(* IEC 61131-3 sources: Bob/Head_Pkg/ValveControl, 14 files *)

(* ---- Types.typ ---- *)
TYPE
	localValve_typ : 	STRUCT
		valveName : STRING[80];
		outputModuleOk : BOOL; (*variable to be linked to the module ok on the IO module used for the outputs*)
		inputModuleOk : BOOL; (*variable to be linked to the module ok on the IO module used for the inputs*)
		doOpen : BOOL; (*variable to be linked to the digital output which opens the valve*)
		doClose : BOOL; (*variable to be linked to the digital output which closes the valve*)
		diOpened : BOOL; (*variable to be linked to the digital input which indicates that the valve is opened*)
		diClosed : BOOL; (*variable to be linked to the digital input which indicates that the valve is closed*)
		position : INT;
		openDebounceTimer : TON;
		closeDebounceTimer : TON;
		openErrorTimer : TON;
		closeErrorTimer : TON;
		MpRecipeRegPar_0 : MpRecipeRegPar;
		MpRecipeRegPar_1 : MpRecipeRegPar;
		openError_r_trig : r_trig;
		closeError_r_trig : r_trig;
		open_and_close_error_r_trig : r_trig;
		io_error_r_trig : r_trig;
		io_error_f_trig : f_trig;
		openAndCloseAlarmID : UDINT;
		closeAlarmID : UDINT;
		openAlarmID : UDINT;
		alarmID : UDINT;
		moduleOKAlarmID : UDINT;
		powerOnTimer : TON;
	END_STRUCT;
END_TYPE

(* ---- balanceTankValve.st ---- *)
ACTION balanceTankAction:

    pCurrentValve ACCESS ADR(gModules[currentModule].heads[currentHead].balanceTank);
    pLocalValve ACCESS ADR(balanceTankValve[indexOf(currentModule, currentHead, NUM_OF_HEADS_PER_MODULE)]);

	IF (pCurrentValve.parameters.machineData.enabled = TRUE) THEN
		IF (pCurrentValve.status.errorActive <> TRUE) THEN

			IF (((pCurrentValve.commands.open = TRUE) AND (pCurrentValve.commands.close = FALSE)) AND
				(pLocalValve.doOpen = FALSE)) THEN
				logDebug(pLocalValve.valveName, 'Module %h, Head %h, Open Command', ADR(logArguments));
				pLocalValve.doOpen := TRUE;
				pLocalValve.doClose := FALSE;
			END_IF

			IF (((pCurrentValve.commands.close = TRUE) AND (pCurrentValve.commands.open = FALSE)) AND
				(pLocalValve.doClose = FALSE)) THEN
				logDebug(pLocalValve.valveName, 'Module %h, Head %h, Close Command', ADR(logArguments));
				pLocalValve.doClose := TRUE;
				pLocalValve.doOpen := FALSE;
			END_IF

			IF (((pCurrentValve.commands.close = FALSE) AND (pCurrentValve.commands.open = FALSE)) AND
				((pLocalValve.doClose <> FALSE) OR (pLocalValve.doOpen <> FALSE))) THEN
				logDebug(pLocalValve.valveName, 'Module %h, Head %h, Center Command', ADR(logArguments));
				pLocalValve.doClose := FALSE;
				pLocalValve.doOpen := FALSE;
			END_IF

		END_IF

		checkValveAlarms;
        updateValveState;

		// 20ms debounce timer
		pLocalValve.openDebounceTimer.IN    := pLocalValve.diOpened;
		pLocalValve.openDebounceTimer.PT    := pCurrentValve.parameters.machineData.debounceTime;
		pLocalValve.openDebounceTimer();

		// 20ms debounce timer
		pLocalValve.closeDebounceTimer.IN := pLocalValve.diClosed;
		pLocalValve.closeDebounceTimer.PT := pCurrentValve.parameters.machineData.debounceTime;
		pLocalValve.closeDebounceTimer();

		pCurrentValve.status.opened             := pLocalValve.openDebounceTimer.Q;
		pCurrentValve.status.closed             := pLocalValve.closeDebounceTimer.Q;
		pCurrentValve.status.centered           := ((pCurrentValve.status.opened <> TRUE) AND (pCurrentValve.status.closed <> TRUE));
		pCurrentValve.status.position           := 0;
		pCurrentValve.status.fullFlowAchieved   := FALSE;

        handleValveErrors;

    END_IF

END_ACTION

(* ---- counterStretchRodValve.st ---- *)
ACTION counterStretchRodAction:

    pCurrentValve ACCESS ADR(gModules[currentModule].heads[currentHead].counterStretchRod );
    pLocalValve ACCESS ADR(counterStretchRodValve[indexOf(currentModule, currentHead, NUM_OF_HEADS_PER_MODULE)]);

	IF (pCurrentValve.parameters.machineData.enabled = TRUE) THEN

		IF (pCurrentValve.status.errorActive <> TRUE) THEN

			IF (((pCurrentValve.commands.open = TRUE) AND (pCurrentValve.commands.close = FALSE)) AND
				(pLocalValve.doOpen = FALSE)) THEN
				logDebug(pLocalValve.valveName, 'Module %h, Head %h, Open Command', ADR(logArguments));
				pLocalValve.doOpen := TRUE;
				pLocalValve.doClose := FALSE;
			END_IF

			IF (((pCurrentValve.commands.close = TRUE) AND (pCurrentValve.commands.open = FALSE)) AND
				(pLocalValve.doClose = FALSE)) THEN
				logDebug(pLocalValve.valveName, 'Module %h, Head %h, Close Command', ADR(logArguments));
				pLocalValve.doClose := TRUE;
				pLocalValve.doOpen := FALSE;
			END_IF

			IF (((pCurrentValve.commands.close = FALSE) AND (pCurrentValve.commands.open = FALSE)) AND
				((pLocalValve.doClose <> FALSE) OR (pLocalValve.doOpen <> FALSE))) THEN
				logDebug(pLocalValve.valveName, 'Module %h, Head %h, Center Command', ADR(logArguments));
				pLocalValve.doClose := FALSE;
				pLocalValve.doOpen := FALSE;
			END_IF

		END_IF

		checkValveAlarms;
        updateValveState;

        // 20ms debounce timer
		pLocalValve.openDebounceTimer.IN    := pLocalValve.diOpened;
		pLocalValve.openDebounceTimer.PT    := pCurrentValve.parameters.machineData.debounceTime;
		pLocalValve.openDebounceTimer();

		// 20ms debounce timer
		pLocalValve.closeDebounceTimer.IN := pLocalValve.diClosed;
		pLocalValve.closeDebounceTimer.PT := pCurrentValve.parameters.machineData.debounceTime;
		pLocalValve.closeDebounceTimer();

		pCurrentValve.status.opened             := pLocalValve.openDebounceTimer.Q;
		pCurrentValve.status.closed             := pLocalValve.closeDebounceTimer.Q;
		pCurrentValve.status.centered           := ((pCurrentValve.status.opened <> TRUE) AND (pCurrentValve.status.closed <> TRUE));
		pCurrentValve.status.position           := 0;
		pCurrentValve.status.fullFlowAchieved   := FALSE;

        handleValveErrors;

	END_IF

END_ACTION

(* ---- cylinderVentValve.st ---- *)
ACTION cylinderVentAction:

    pCurrentValve ACCESS ADR(gModules[currentModule].heads[currentHead].cylinderVent);
    pLocalValve ACCESS ADR(cylinderVentValve[indexOf(currentModule, currentHead, NUM_OF_HEADS_PER_MODULE)]);

	IF (pCurrentValve.parameters.machineData.enabled = TRUE) THEN

		IF (pCurrentValve.status.errorActive <> TRUE) THEN

			IF (((pCurrentValve.commands.open = TRUE) AND (pCurrentValve.commands.close = FALSE)) AND
				(pLocalValve.doOpen = FALSE)) THEN
				logDebug('Cylinder Vent Valve', 'Module %h, Head %h, Open Command', ADR(logArguments));
				pLocalValve.doOpen := TRUE;
				pLocalValve.doClose := FALSE;
			END_IF

			IF (((pCurrentValve.commands.close = TRUE) AND (pCurrentValve.commands.open = FALSE)) AND
				(pLocalValve.doClose = FALSE)) THEN
				logDebug('Cylinder Vent Valve', 'Module %h, Head %h, Close Command', ADR(logArguments));
				pLocalValve.doClose := TRUE;
				pLocalValve.doOpen := FALSE;
			END_IF

			IF (((pCurrentValve.commands.close = FALSE) AND (pCurrentValve.commands.open = FALSE)) AND
				((pLocalValve.doClose <> FALSE) OR (pLocalValve.doOpen <> FALSE))) THEN
				logDebug('Cylinder Vent Valve', 'Module %h, Head %h, Center Command', ADR(logArguments));
				pLocalValve.doClose := FALSE;
				pLocalValve.doOpen := FALSE;
			END_IF

		END_IF

        checkValveAlarms;
        updateValveState;

		// 20ms debounce timer
		pLocalValve.openDebounceTimer.IN    := pLocalValve.diOpened;
		pLocalValve.openDebounceTimer.PT    := pCurrentValve.parameters.machineData.debounceTime;
		pLocalValve.openDebounceTimer();

		// 20ms debounce timer
		pLocalValve.closeDebounceTimer.IN := pLocalValve.diClosed;
		pLocalValve.closeDebounceTimer.PT := pCurrentValve.parameters.machineData.debounceTime;
		pLocalValve.closeDebounceTimer();

		pCurrentValve.status.opened             := pLocalValve.openDebounceTimer.Q;
		pCurrentValve.status.closed             := pLocalValve.closeDebounceTimer.Q;
		pCurrentValve.status.centered           := ((pCurrentValve.status.opened <> TRUE) AND (pCurrentValve.status.closed <> TRUE));
		pCurrentValve.status.position           := 0;
		pCurrentValve.status.fullFlowAchieved   := FALSE;

        handleValveErrors;

	END_IF

END_ACTION

(* ---- fillLevelCylinderValve.st ---- *)
ACTION fillLevelCylinderValveAction:

    pCurrentValve ACCESS ADR(gModules[currentModule].heads[currentHead].fillLevelCylinderValve);
    pLocalValve ACCESS ADR(fillLevelCylinderValve[indexOf(currentModule, currentHead, NUM_OF_HEADS_PER_MODULE)]);

	IF (pCurrentValve.parameters.machineData.enabled = TRUE) THEN

		IF (pCurrentValve.status.errorActive <> TRUE) THEN

			IF (((pCurrentValve.commands.open = TRUE) AND (pCurrentValve.commands.close = FALSE)) AND
				(pLocalValve.doOpen = FALSE)) THEN
				logDebug(pLocalValve.valveName, 'Module %h, Head %h, Retract Command', ADR(logArguments));
				pLocalValve.doOpen := TRUE;
				pLocalValve.doClose := FALSE;
			END_IF

			IF (((pCurrentValve.commands.close = TRUE) AND (pCurrentValve.commands.open = FALSE)) AND
				(pLocalValve.doClose = FALSE)) THEN
				logDebug(pLocalValve.valveName, 'Module %h, Head %h, Extend Command', ADR(logArguments));
				pLocalValve.doClose := TRUE;
				pLocalValve.doOpen := FALSE;
			END_IF

			IF (((pCurrentValve.commands.close = FALSE) AND (pCurrentValve.commands.open = FALSE)) AND
				((pLocalValve.doClose <> FALSE) OR (pLocalValve.doOpen <> FALSE))) THEN
				logDebug(pLocalValve.valveName, 'Module %h, Head %h, Center Command', ADR(logArguments));
				pLocalValve.doClose := FALSE;
				pLocalValve.doOpen := FALSE;
			END_IF

		END_IF

        checkValveAlarms;
        updateValveState;

		// 20ms debounce timer
		pLocalValve.openDebounceTimer.IN    := pLocalValve.diOpened;
		pLocalValve.openDebounceTimer.PT    := pCurrentValve.parameters.machineData.debounceTime;
		pLocalValve.openDebounceTimer();

		// 20ms debounce timer
		pLocalValve.closeDebounceTimer.IN := pLocalValve.diClosed;
		pLocalValve.closeDebounceTimer.PT := pCurrentValve.parameters.machineData.debounceTime;
		pLocalValve.closeDebounceTimer();

		pCurrentValve.status.opened             := pLocalValve.openDebounceTimer.Q;
		pCurrentValve.status.closed             := pLocalValve.closeDebounceTimer.Q;
		pCurrentValve.status.centered           := ((pCurrentValve.status.opened <> TRUE) AND (pCurrentValve.status.closed <> TRUE));
		pCurrentValve.status.position           := 0;
		pCurrentValve.status.fullFlowAchieved   := FALSE;

        handleValveErrors;

	END_IF

END_ACTION

(* ---- fillLevelDrainValve.st ---- *)
ACTION fillLevelDrainValveAction:

    pCurrentValve ACCESS ADR(gModules[currentModule].heads[currentHead].fillLevelDrainValve);
    pLocalValve ACCESS ADR(fillLevelDrainValve[indexOf(currentModule, currentHead, NUM_OF_HEADS_PER_MODULE)]);

	IF (pCurrentValve.parameters.machineData.enabled = TRUE) THEN

		IF (pCurrentValve.status.errorActive <> TRUE) THEN

			IF (((pCurrentValve.commands.open = TRUE) AND (pCurrentValve.commands.close = FALSE)) AND
				(pLocalValve.doOpen = FALSE)) THEN
				logDebug(pLocalValve.valveName, 'Module %h, Head %h, Open Command', ADR(logArguments));
				pLocalValve.doOpen := TRUE;
				pLocalValve.doClose := FALSE;
			END_IF

			IF (((pCurrentValve.commands.close = TRUE) AND (pCurrentValve.commands.open = FALSE)) AND
				(pLocalValve.doClose = FALSE)) THEN
				logDebug(pLocalValve.valveName, 'Module %h, Head %h, Close Command', ADR(logArguments));
				pLocalValve.doClose := TRUE;
				pLocalValve.doOpen := FALSE;
			END_IF

			IF (((pCurrentValve.commands.close = FALSE) AND (pCurrentValve.commands.open = FALSE)) AND
				((pLocalValve.doClose <> FALSE) OR (pLocalValve.doOpen <> FALSE))) THEN
				logDebug(pLocalValve.valveName, 'Module %h, Head %h, Center Command', ADR(logArguments));
				pLocalValve.doClose := FALSE;
				pLocalValve.doOpen := FALSE;
			END_IF

		END_IF

        checkValveAlarms;
        updateValveState;

		// 20ms debounce timer
		pLocalValve.openDebounceTimer.IN    := pLocalValve.diOpened;
		pLocalValve.openDebounceTimer.PT    := pCurrentValve.parameters.machineData.debounceTime;
		pLocalValve.openDebounceTimer();

		// 20ms debounce timer
		pLocalValve.closeDebounceTimer.IN := pLocalValve.diClosed;
		pLocalValve.closeDebounceTimer.PT := pCurrentValve.parameters.machineData.debounceTime;
		pLocalValve.closeDebounceTimer();

		pCurrentValve.status.opened             := pLocalValve.openDebounceTimer.Q;
		pCurrentValve.status.closed             := pLocalValve.closeDebounceTimer.Q;
		pCurrentValve.status.centered           := ((pCurrentValve.status.opened <> TRUE) AND (pCurrentValve.status.closed <> TRUE));
		pCurrentValve.status.position           := 0;
		pCurrentValve.status.fullFlowAchieved   := FALSE;

        handleValveErrors;

	END_IF

END_ACTION

(* ---- fillLevelSuctionValve.st ---- *)
ACTION fillLevelSuctionValveAction:

    pCurrentValve ACCESS ADR(gModules[currentModule].heads[currentHead].fillLevelSuctionValve);
    pLocalValve ACCESS ADR(fillLevelSuctionValve[indexOf(currentModule, currentHead, NUM_OF_HEADS_PER_MODULE)]);

	IF (pCurrentValve.parameters.machineData.enabled = TRUE) THEN

		IF (pCurrentValve.status.errorActive <> TRUE) THEN

			IF (((pCurrentValve.commands.open = TRUE) AND (pCurrentValve.commands.close = FALSE)) AND
				(pLocalValve.doOpen = FALSE)) THEN
				logDebug(pLocalValve.valveName, 'Module %h, Head %h, Open Command', ADR(logArguments));
				pLocalValve.doOpen := TRUE;
				pLocalValve.doClose := FALSE;
			END_IF

			IF (((pCurrentValve.commands.close = TRUE) AND (pCurrentValve.commands.open = FALSE)) AND
				(pLocalValve.doClose = FALSE)) THEN
				logDebug(pLocalValve.valveName, 'Module %h, Head %h, Close Command', ADR(logArguments));
				pLocalValve.doClose := TRUE;
				pLocalValve.doOpen := FALSE;
			END_IF

			IF (((pCurrentValve.commands.close = FALSE) AND (pCurrentValve.commands.open = FALSE)) AND
				((pLocalValve.doClose <> FALSE) OR (pLocalValve.doOpen <> FALSE))) THEN
				logDebug(pLocalValve.valveName, 'Module %h, Head %h, Center Command', ADR(logArguments));
				pLocalValve.doClose := FALSE;
				pLocalValve.doOpen := FALSE;
			END_IF

        END_IF

        checkValveAlarms;
        updateValveState;

		// 20ms debounce timer
		pLocalValve.openDebounceTimer.IN    := pLocalValve.diOpened;
		pLocalValve.openDebounceTimer.PT    := pCurrentValve.parameters.machineData.debounceTime;
		pLocalValve.openDebounceTimer();

		// 20ms debounce timer
		pLocalValve.closeDebounceTimer.IN := pLocalValve.diClosed;
		pLocalValve.closeDebounceTimer.PT := pCurrentValve.parameters.machineData.debounceTime;
		pLocalValve.closeDebounceTimer();

		pCurrentValve.status.opened             := pLocalValve.openDebounceTimer.Q;
		pCurrentValve.status.closed             := pLocalValve.closeDebounceTimer.Q;
		pCurrentValve.status.centered           := ((pCurrentValve.status.opened <> TRUE) AND (pCurrentValve.status.closed <> TRUE));
		pCurrentValve.status.position           := 0;
		pCurrentValve.status.fullFlowAchieved   := FALSE;

        handleValveErrors;

	END_IF

END_ACTION

(* ---- fillValve.st ---- *)
ACTION fillAction:

	pCurrentValve ACCESS ADR(gModules[currentModule].heads[currentHead].fillValve);
	pLocalValve ACCESS ADR(fillValve[indexOf(currentModule, currentHead, NUM_OF_HEADS_PER_MODULE)]);

	IF (pCurrentValve.parameters.machineData.enabled = TRUE) THEN

		IF (pCurrentValve.status.errorActive <> TRUE) THEN

			IF (((pCurrentValve.commands.open = TRUE) AND (pCurrentValve.commands.close = FALSE)) AND
				(pLocalValve.doOpen = FALSE)) THEN
				logDebug(pLocalValve.valveName, 'Module %h, Head %h, Open Command', ADR(logArguments));
				pLocalValve.doOpen := TRUE;
				pLocalValve.doClose := FALSE;

			END_IF

			IF (((pCurrentValve.commands.close = TRUE) AND (pCurrentValve.commands.open = FALSE)) AND
				(pLocalValve.doClose = FALSE)) THEN
				logDebug(pLocalValve.valveName, 'Module %h, Head %h, Close Command', ADR(logArguments));
				pLocalValve.doClose := TRUE;
				pLocalValve.doOpen := FALSE;
			END_IF

			IF (((pCurrentValve.commands.close = FALSE) AND (pCurrentValve.commands.open = FALSE)) AND
				((pLocalValve.doClose <> FALSE) OR (pLocalValve.doOpen <> FALSE))) THEN
				logDebug(pLocalValve.valveName, 'Module %h, Head %h, Center Command', ADR(logArguments));
				pLocalValve.doClose := FALSE;
				pLocalValve.doOpen := FALSE;
			END_IF

		END_IF

        checkValveAlarms;
        updateValveState;

		// 20ms debounce timer
		pLocalValve.openDebounceTimer.IN    := pLocalValve.diOpened;
		pLocalValve.openDebounceTimer.PT    := pCurrentValve.parameters.machineData.debounceTime;
		pLocalValve.openDebounceTimer();

		// 20ms debounce timer
		pLocalValve.closeDebounceTimer.IN := pLocalValve.diClosed;
		pLocalValve.closeDebounceTimer.PT := pCurrentValve.parameters.machineData.debounceTime;
		pLocalValve.closeDebounceTimer();

		pCurrentValve.status.opened             := pLocalValve.openDebounceTimer.Q;
		pCurrentValve.status.closed             := pLocalValve.closeDebounceTimer.Q;
		pCurrentValve.status.centered           := ((pCurrentValve.status.opened <> TRUE) AND (pCurrentValve.status.closed <> TRUE));
		pCurrentValve.status.position           := 0;
		pCurrentValve.status.fullFlowAchieved   := FALSE;

        handleValveErrors;

	END_IF

END_ACTION

(* ---- formingValve.st ---- *)
ACTION formingValveAction:

    pCurrentValve ACCESS ADR(gModules[currentModule].heads[currentHead].formingValve);
    pLocalValve ACCESS ADR(formingValve[indexOf(currentModule, currentHead, NUM_OF_HEADS_PER_MODULE)]);

	IF (pCurrentValve.parameters.machineData.enabled = TRUE) THEN

		IF (pCurrentValve.status.errorActive <> TRUE) THEN

			IF (((pCurrentValve.commands.open = TRUE) AND (pCurrentValve.commands.close = FALSE)) AND
				(pLocalValve.doOpen = FALSE)) THEN
				logDebug(pLocalValve.valveName, 'Module %h, Head %h, Open Command', ADR(logArguments));
				pLocalValve.doOpen := TRUE;
				pLocalValve.doClose := FALSE;
			END_IF

			IF (((pCurrentValve.commands.close = TRUE) AND (pCurrentValve.commands.open = FALSE)) AND
				(pLocalValve.doClose = FALSE)) THEN
				logDebug(pLocalValve.valveName, 'Module %h, Head %h, Close Command', ADR(logArguments));
				pLocalValve.doClose := TRUE;
				pLocalValve.doOpen := FALSE;
			END_IF

			IF (((pCurrentValve.commands.close = FALSE) AND (pCurrentValve.commands.open = FALSE)) AND
				((pLocalValve.doClose <> FALSE) OR (pLocalValve.doOpen <> FALSE))) THEN
				logDebug(pLocalValve.valveName, 'Module %h, Head %h, Center Command', ADR(logArguments));
				pLocalValve.doClose := FALSE;
				pLocalValve.doOpen := FALSE;
			END_IF

		END_IF

        checkValveAlarms;
        updateValveState;

		// 20ms debounce timer
		pLocalValve.openDebounceTimer.IN    := pLocalValve.diOpened;
		pLocalValve.openDebounceTimer.PT    := pCurrentValve.parameters.machineData.debounceTime;
		pLocalValve.openDebounceTimer();

		// 20ms debounce timer
		pLocalValve.closeDebounceTimer.IN := pLocalValve.diClosed;
		pLocalValve.closeDebounceTimer.PT := pCurrentValve.parameters.machineData.debounceTime;
		pLocalValve.closeDebounceTimer();

		pCurrentValve.status.opened         := pLocalValve.openDebounceTimer.Q;
		pCurrentValve.status.closed         := pLocalValve.closeDebounceTimer.Q;
		pCurrentValve.status.centered       := ((pCurrentValve.status.opened <> TRUE) AND (pCurrentValve.status.closed <> TRUE));
		pCurrentValve.status.position       := 0;

        handleValveErrors;

	END_IF

END_ACTION

(* ---- Main.st ---- *)
PROGRAM _INIT

    // register the balance tank parameters
    gModules[0].heads[0].balanceTank;
    balanceTankValve[0].MpRecipeRegPar_0.PVName := ADR('gModules[0].heads[0].balanceTank.parameters.machineData');
    balanceTankValve[1].MpRecipeRegPar_0.PVName := ADR('gModules[0].heads[1].balanceTank.parameters.machineData');
    balanceTankValve[2].MpRecipeRegPar_0.PVName := ADR('gModules[1].heads[0].balanceTank.parameters.machineData');
    balanceTankValve[3].MpRecipeRegPar_0.PVName := ADR('gModules[1].heads[1].balanceTank.parameters.machineData');

    FOR currentHead:=0 TO NUMBER_OF_HEADS_M1 DO
        balanceTankValve[currentHead].MpRecipeRegPar_0.MpLink := ADR(gMachineRecipe);
        balanceTankValve[currentHead].MpRecipeRegPar_0.Enable := TRUE;
        balanceTankValve[currentHead].MpRecipeRegPar_0.Category := ADR(MACHINE_CATEGORY);
        balanceTankValve[currentHead].MpRecipeRegPar_0();
    END_FOR

    balanceTankValve[0].MpRecipeRegPar_1.PVName := ADR('gModules[0].heads[0].balanceTank.parameters.processData');
    balanceTankValve[1].MpRecipeRegPar_1.PVName := ADR('gModules[0].heads[1].balanceTank.parameters.processData');
    balanceTankValve[2].MpRecipeRegPar_1.PVName := ADR('gModules[1].heads[0].balanceTank.parameters.processData');
    balanceTankValve[3].MpRecipeRegPar_1.PVName := ADR('gModules[1].heads[1].balanceTank.parameters.processData');

    FOR currentHead:=0 TO NUMBER_OF_HEADS_M1 DO
        balanceTankValve[currentHead].MpRecipeRegPar_1.MpLink := ADR(gProcessRecipe);
        balanceTankValve[currentHead].MpRecipeRegPar_1.Enable := TRUE;
        balanceTankValve[currentHead].MpRecipeRegPar_1.Category := ADR(PROCESS_CATEGORY);
        balanceTankValve[currentHead].MpRecipeRegPar_1();
    END_FOR

    // register the fill valve parameters
    gModules[0].heads[0].fillValve;
    fillValve[0].MpRecipeRegPar_0.PVName := ADR('gModules[0].heads[0].fillValve.parameters.machineData');
    fillValve[1].MpRecipeRegPar_0.PVName := ADR('gModules[0].heads[1].fillValve.parameters.machineData');
    fillValve[2].MpRecipeRegPar_0.PVName := ADR('gModules[1].heads[0].fillValve.parameters.machineData');
    fillValve[3].MpRecipeRegPar_0.PVName := ADR('gModules[1].heads[1].fillValve.parameters.machineData');

    FOR currentHead:=0 TO NUMBER_OF_HEADS_M1 DO
        fillValve[currentHead].MpRecipeRegPar_0.MpLink := ADR(gMachineRecipe);
        fillValve[currentHead].MpRecipeRegPar_0.Enable := TRUE;
        fillValve[currentHead].MpRecipeRegPar_0.Category := ADR(MACHINE_CATEGORY);
        fillValve[currentHead].MpRecipeRegPar_0();
    END_FOR

    fillValve[0].MpRecipeRegPar_1.PVName := ADR('gModules[0].heads[0].fillValve.parameters.processData');
    fillValve[1].MpRecipeRegPar_1.PVName := ADR('gModules[0].heads[1].fillValve.parameters.processData');
    fillValve[2].MpRecipeRegPar_1.PVName := ADR('gModules[1].heads[0].fillValve.parameters.processData');
    fillValve[3].MpRecipeRegPar_1.PVName := ADR('gModules[1].heads[1].fillValve.parameters.processData');

    FOR currentHead:=0 TO NUMBER_OF_HEADS_M1 DO
        fillValve[currentHead].MpRecipeRegPar_1.MpLink := ADR(gProcessRecipe);
        fillValve[currentHead].MpRecipeRegPar_1.Enable := TRUE;
        fillValve[currentHead].MpRecipeRegPar_1.Category := ADR(PROCESS_CATEGORY);
        fillValve[currentHead].MpRecipeRegPar_1();
    END_FOR

    // register the fill vent parameters
    gModules[0].heads[0].cylinderVent;
    cylinderVentValve[0].MpRecipeRegPar_0.PVName := ADR('gModules[0].heads[0].cylinderVent.parameters.machineData');
    cylinderVentValve[1].MpRecipeRegPar_0.PVName := ADR('gModules[0].heads[1].cylinderVent.parameters.machineData');
    cylinderVentValve[2].MpRecipeRegPar_0.PVName := ADR('gModules[1].heads[0].cylinderVent.parameters.machineData');
    cylinderVentValve[3].MpRecipeRegPar_0.PVName := ADR('gModules[1].heads[1].cylinderVent.parameters.machineData');

    FOR currentHead:=0 TO NUMBER_OF_HEADS_M1 DO
        cylinderVentValve[currentHead].MpRecipeRegPar_0.MpLink := ADR(gMachineRecipe);
        cylinderVentValve[currentHead].MpRecipeRegPar_0.Enable := TRUE;
        cylinderVentValve[currentHead].MpRecipeRegPar_0.Category := ADR(MACHINE_CATEGORY);
        cylinderVentValve[currentHead].MpRecipeRegPar_0();
    END_FOR

    cylinderVentValve[0].MpRecipeRegPar_1.PVName := ADR('gModules[0].heads[0].cylinderVent.parameters.processData');
    cylinderVentValve[1].MpRecipeRegPar_1.PVName := ADR('gModules[0].heads[1].cylinderVent.parameters.processData');
    cylinderVentValve[2].MpRecipeRegPar_1.PVName := ADR('gModules[1].heads[0].cylinderVent.parameters.processData');
    cylinderVentValve[3].MpRecipeRegPar_1.PVName := ADR('gModules[1].heads[1].cylinderVent.parameters.processData');

    FOR currentHead:=0 TO NUMBER_OF_HEADS_M1 DO
        cylinderVentValve[currentHead].MpRecipeRegPar_1.MpLink := ADR(gProcessRecipe);
        cylinderVentValve[currentHead].MpRecipeRegPar_1.Enable := TRUE;
        cylinderVentValve[currentHead].MpRecipeRegPar_1.Category := ADR(PROCESS_CATEGORY);
        cylinderVentValve[currentHead].MpRecipeRegPar_1();
    END_FOR

    // register the nozzle parameters
    gModules[0].heads[0].nozzle;
    nozzleValve[0].MpRecipeRegPar_0.PVName := ADR('gModules[0].heads[0].nozzle.parameters.machineData');
    nozzleValve[1].MpRecipeRegPar_0.PVName := ADR('gModules[0].heads[1].nozzle.parameters.machineData');
    nozzleValve[2].MpRecipeRegPar_0.PVName := ADR('gModules[1].heads[0].nozzle.parameters.machineData');
    nozzleValve[3].MpRecipeRegPar_0.PVName := ADR('gModules[1].heads[1].nozzle.parameters.machineData');

    FOR currentHead:=0 TO NUMBER_OF_HEADS_M1 DO
        nozzleValve[currentHead].MpRecipeRegPar_0.MpLink := ADR(gMachineRecipe);
        nozzleValve[currentHead].MpRecipeRegPar_0.Enable := TRUE;
        nozzleValve[currentHead].MpRecipeRegPar_0.Category := ADR(MACHINE_CATEGORY);
        nozzleValve[currentHead].MpRecipeRegPar_0();
    END_FOR

    nozzleValve[0].MpRecipeRegPar_1.PVName := ADR('gModules[0].heads[0].nozzle.parameters.processData');
    nozzleValve[1].MpRecipeRegPar_1.PVName := ADR('gModules[0].heads[1].nozzle.parameters.processData');
    nozzleValve[2].MpRecipeRegPar_1.PVName := ADR('gModules[1].heads[0].nozzle.parameters.processData');
    nozzleValve[3].MpRecipeRegPar_1.PVName := ADR('gModules[1].heads[1].nozzle.parameters.processData');

    FOR currentHead:=0 TO NUMBER_OF_HEADS_M1 DO
        nozzleValve[currentHead].MpRecipeRegPar_1.MpLink := ADR(gProcessRecipe);
        nozzleValve[currentHead].MpRecipeRegPar_1.Enable := TRUE;
        nozzleValve[currentHead].MpRecipeRegPar_1.Category := ADR(PROCESS_CATEGORY);
        nozzleValve[currentHead].MpRecipeRegPar_1();
    END_FOR

    // register the recirculationValve parameters
    gModules[0].heads[0].recirculationValve;
    recirculationValve[0].MpRecipeRegPar_0.PVName := ADR('gModules[0].heads[0].recirculationValve.parameters.machineData');
    recirculationValve[1].MpRecipeRegPar_0.PVName := ADR('gModules[0].heads[1].recirculationValve.parameters.machineData');
    recirculationValve[2].MpRecipeRegPar_0.PVName := ADR('gModules[1].heads[0].recirculationValve.parameters.machineData');
    recirculationValve[3].MpRecipeRegPar_0.PVName := ADR('gModules[1].heads[1].recirculationValve.parameters.machineData');

    FOR currentHead:=0 TO NUMBER_OF_HEADS_M1 DO
        recirculationValve[currentHead].MpRecipeRegPar_0.MpLink := ADR(gMachineRecipe);
        recirculationValve[currentHead].MpRecipeRegPar_0.Enable := TRUE;
        recirculationValve[currentHead].MpRecipeRegPar_0.Category := ADR(MACHINE_CATEGORY);
        recirculationValve[currentHead].MpRecipeRegPar_0();
    END_FOR

    recirculationValve[0].MpRecipeRegPar_1.PVName := ADR('gModules[0].heads[0].recirculationValve.parameters.processData');
    recirculationValve[1].MpRecipeRegPar_1.PVName := ADR('gModules[0].heads[1].recirculationValve.parameters.processData');
    recirculationValve[2].MpRecipeRegPar_1.PVName := ADR('gModules[1].heads[0].recirculationValve.parameters.processData');
    recirculationValve[3].MpRecipeRegPar_1.PVName := ADR('gModules[1].heads[1].recirculationValve.parameters.processData');

    FOR currentHead:=0 TO NUMBER_OF_HEADS_M1 DO
        recirculationValve[currentHead].MpRecipeRegPar_1.MpLink := ADR(gProcessRecipe);
        recirculationValve[currentHead].MpRecipeRegPar_1.Enable := TRUE;
        recirculationValve[currentHead].MpRecipeRegPar_1.Category := ADR(PROCESS_CATEGORY);
        recirculationValve[currentHead].MpRecipeRegPar_1();
    END_FOR

    // register the sealPin parameters
    gModules[0].heads[0].sealPin;
    sealPinValve[0].MpRecipeRegPar_0.PVName := ADR('gModules[0].heads[0].sealPin.parameters.machineData');
    sealPinValve[1].MpRecipeRegPar_0.PVName := ADR('gModules[0].heads[1].sealPin.parameters.machineData');
    sealPinValve[2].MpRecipeRegPar_0.PVName := ADR('gModules[1].heads[0].sealPin.parameters.machineData');
    sealPinValve[3].MpRecipeRegPar_0.PVName := ADR('gModules[1].heads[1].sealPin.parameters.machineData');

    FOR currentHead:=0 TO NUMBER_OF_HEADS_M1 DO
        sealPinValve[currentHead].MpRecipeRegPar_0.MpLink := ADR(gMachineRecipe);
        sealPinValve[currentHead].MpRecipeRegPar_0.Enable := TRUE;
        sealPinValve[currentHead].MpRecipeRegPar_0.Category := ADR(MACHINE_CATEGORY);
        sealPinValve[currentHead].MpRecipeRegPar_0();
    END_FOR

    sealPinValve[0].MpRecipeRegPar_1.PVName := ADR('gModules[0].heads[0].sealPin.parameters.processData');
    sealPinValve[1].MpRecipeRegPar_1.PVName := ADR('gModules[0].heads[1].sealPin.parameters.processData');
    sealPinValve[2].MpRecipeRegPar_1.PVName := ADR('gModules[1].heads[0].sealPin.parameters.processData');
    sealPinValve[3].MpRecipeRegPar_1.PVName := ADR('gModules[1].heads[1].sealPin.parameters.processData');

    FOR currentHead:=0 TO NUMBER_OF_HEADS_M1 DO
        sealPinValve[currentHead].MpRecipeRegPar_1.MpLink := ADR(gProcessRecipe);
        sealPinValve[currentHead].MpRecipeRegPar_1.Enable := TRUE;
        sealPinValve[currentHead].MpRecipeRegPar_1.Category := ADR(PROCESS_CATEGORY);
        sealPinValve[currentHead].MpRecipeRegPar_1();
    END_FOR

    // register the sealPin parameters
    gModules[0].heads[0].sealPin;
    counterStretchRodValve[0].MpRecipeRegPar_0.PVName := ADR('gModules[0].heads[0].counterStretchRod.parameters.machineData');
    counterStretchRodValve[1].MpRecipeRegPar_0.PVName := ADR('gModules[0].heads[1].counterStretchRod.parameters.machineData');
    counterStretchRodValve[2].MpRecipeRegPar_0.PVName := ADR('gModules[1].heads[0].counterStretchRod.parameters.machineData');
    counterStretchRodValve[3].MpRecipeRegPar_0.PVName := ADR('gModules[1].heads[1].counterStretchRod.parameters.machineData');

    FOR currentHead:=0 TO NUMBER_OF_HEADS_M1 DO
        counterStretchRodValve[currentHead].MpRecipeRegPar_0.MpLink := ADR(gMachineRecipe);
        counterStretchRodValve[currentHead].MpRecipeRegPar_0.Enable := TRUE;
        counterStretchRodValve[currentHead].MpRecipeRegPar_0.Category := ADR(MACHINE_CATEGORY);
        counterStretchRodValve[currentHead].MpRecipeRegPar_0();
    END_FOR

    counterStretchRodValve[0].MpRecipeRegPar_1.PVName := ADR('gModules[0].heads[0].counterStretchRod.parameters.processData');
    counterStretchRodValve[1].MpRecipeRegPar_1.PVName := ADR('gModules[0].heads[1].counterStretchRod.parameters.processData');
    counterStretchRodValve[2].MpRecipeRegPar_1.PVName := ADR('gModules[1].heads[0].counterStretchRod.parameters.processData');
    counterStretchRodValve[3].MpRecipeRegPar_1.PVName := ADR('gModules[1].heads[1].counterStretchRod.parameters.processData');

    FOR currentHead:=0 TO NUMBER_OF_HEADS_M1 DO
        counterStretchRodValve[currentHead].MpRecipeRegPar_1.MpLink := ADR(gProcessRecipe);
        counterStretchRodValve[currentHead].MpRecipeRegPar_1.Enable := TRUE;
        counterStretchRodValve[currentHead].MpRecipeRegPar_1.Category := ADR(PROCESS_CATEGORY);
        counterStretchRodValve[currentHead].MpRecipeRegPar_1();
    END_FOR

    // register the forming valve parameters
    gModules[0].heads[0].formingValve;
    formingValve[0].MpRecipeRegPar_0.PVName := ADR('gModules[0].heads[0].formingValve.parameters.machineData');
    formingValve[1].MpRecipeRegPar_0.PVName := ADR('gModules[0].heads[1].formingValve.parameters.machineData');
    formingValve[2].MpRecipeRegPar_0.PVName := ADR('gModules[1].heads[0].formingValve.parameters.machineData');
    formingValve[3].MpRecipeRegPar_0.PVName := ADR('gModules[1].heads[1].formingValve.parameters.machineData');

    FOR currentHead:=0 TO NUMBER_OF_HEADS_M1 DO
        formingValve[currentHead].MpRecipeRegPar_0.MpLink := ADR(gMachineRecipe);
        formingValve[currentHead].MpRecipeRegPar_0.Enable := TRUE;
        formingValve[currentHead].MpRecipeRegPar_0.Category := ADR(MACHINE_CATEGORY);
        formingValve[currentHead].MpRecipeRegPar_0();
    END_FOR

    formingValve[0].MpRecipeRegPar_1.PVName := ADR('gModules[0].heads[0].formingValve.parameters.processData');
    formingValve[1].MpRecipeRegPar_1.PVName := ADR('gModules[0].heads[1].formingValve.parameters.processData');
    formingValve[2].MpRecipeRegPar_1.PVName := ADR('gModules[1].heads[0].formingValve.parameters.processData');
    formingValve[3].MpRecipeRegPar_1.PVName := ADR('gModules[1].heads[1].formingValve.parameters.processData');

    FOR currentHead:=0 TO NUMBER_OF_HEADS_M1 DO
        formingValve[currentHead].MpRecipeRegPar_1.MpLink := ADR(gProcessRecipe);
        formingValve[currentHead].MpRecipeRegPar_1.Enable := TRUE;
        formingValve[currentHead].MpRecipeRegPar_1.Category := ADR(PROCESS_CATEGORY);
        formingValve[currentHead].MpRecipeRegPar_1();
	END_FOR

	// register the FillLevel Cyclinder valve parameters
	gModules[0].heads[0].fillLevelCylinderValve;
	fillLevelCylinderValve[0].MpRecipeRegPar_0.PVName := ADR('gModules[0].heads[0]fillLevelCylinderValve.parameters.machineData');
	fillLevelCylinderValve[1].MpRecipeRegPar_0.PVName := ADR('gModules[0].heads[1].fillLevelCylinderValve.parameters.machineData');
	fillLevelCylinderValve[2].MpRecipeRegPar_0.PVName := ADR('gModules[1].heads[0].fillLevelCylinderValve.parameters.machineData');
	fillLevelCylinderValve[3].MpRecipeRegPar_0.PVName := ADR('gModules[1].heads[1].fillLevelCylinderValve.parameters.machineData');

	FOR currentHead:=0 TO NUMBER_OF_HEADS_M1 DO
		fillLevelCylinderValve[currentHead].MpRecipeRegPar_0.MpLink := ADR(gMachineRecipe);
		fillLevelCylinderValve[currentHead].MpRecipeRegPar_0.Enable := TRUE;
		fillLevelCylinderValve[currentHead].MpRecipeRegPar_0.Category := ADR(MACHINE_CATEGORY);
		fillLevelCylinderValve[currentHead].MpRecipeRegPar_0();
	END_FOR

	fillLevelCylinderValve[0].MpRecipeRegPar_1.PVName := ADR('gModules[0].heads[0].fillLevelCylinderValve.parameters.processData');
	fillLevelCylinderValve[1].MpRecipeRegPar_1.PVName := ADR('gModules[0].heads[1].fillLevelCylinderValve.parameters.processData');
	fillLevelCylinderValve[2].MpRecipeRegPar_1.PVName := ADR('gModules[1].heads[0].fillLevelCylinderValve.parameters.processData');
	fillLevelCylinderValve[3].MpRecipeRegPar_1.PVName := ADR('gModules[1].heads[1].fillLevelCylinderValve.parameters.processData');

	FOR currentHead:=0 TO NUMBER_OF_HEADS_M1 DO
		fillLevelCylinderValve[currentHead].MpRecipeRegPar_1.MpLink := ADR(gProcessRecipe);
		fillLevelCylinderValve[currentHead].MpRecipeRegPar_1.Enable := TRUE;
		fillLevelCylinderValve[currentHead].MpRecipeRegPar_1.Category := ADR(PROCESS_CATEGORY);
		fillLevelCylinderValve[currentHead].MpRecipeRegPar_1();
	END_FOR

	// register the FillLevel Suction valve parameters
	gModules[0].heads[0].fillLevelCylinderValve;
	fillLevelSuctionValve[0].MpRecipeRegPar_0.PVName := ADR('gModules[0].heads[0]fillLevelSuctionValve.parameters.machineData');
	fillLevelSuctionValve[1].MpRecipeRegPar_0.PVName := ADR('gModules[0].heads[1].fillLevelSuctionValve.parameters.machineData');
	fillLevelSuctionValve[2].MpRecipeRegPar_0.PVName := ADR('gModules[1].heads[0].fillLevelSuctionValve.parameters.machineData');
	fillLevelSuctionValve[3].MpRecipeRegPar_0.PVName := ADR('gModules[1].heads[1].fillLevelSuctionValve.parameters.machineData');

	FOR currentHead:=0 TO NUMBER_OF_HEADS_M1 DO
		fillLevelSuctionValve[currentHead].MpRecipeRegPar_0.MpLink := ADR(gMachineRecipe);
		fillLevelSuctionValve[currentHead].MpRecipeRegPar_0.Enable := TRUE;
		fillLevelSuctionValve[currentHead].MpRecipeRegPar_0.Category := ADR(MACHINE_CATEGORY);
		fillLevelSuctionValve[currentHead].MpRecipeRegPar_0();
	END_FOR

	fillLevelSuctionValve[0].MpRecipeRegPar_1.PVName := ADR('gModules[0].heads[0].fillLevelSuctionValve.parameters.processData');
	fillLevelSuctionValve[1].MpRecipeRegPar_1.PVName := ADR('gModules[0].heads[1].fillLevelSuctionValve.parameters.processData');
	fillLevelSuctionValve[2].MpRecipeRegPar_1.PVName := ADR('gModules[1].heads[0].fillLevelSuctionValve.parameters.processData');
	fillLevelSuctionValve[3].MpRecipeRegPar_1.PVName := ADR('gModules[1].heads[1].fillLevelSuctionValve.parameters.processData');

	FOR currentHead:=0 TO NUMBER_OF_HEADS_M1 DO
		fillLevelSuctionValve[currentHead].MpRecipeRegPar_1.MpLink := ADR(gProcessRecipe);
		fillLevelSuctionValve[currentHead].MpRecipeRegPar_1.Enable := TRUE;
		fillLevelSuctionValve[currentHead].MpRecipeRegPar_1.Category := ADR(PROCESS_CATEGORY);
		fillLevelSuctionValve[currentHead].MpRecipeRegPar_1();
	END_FOR

	// register the FillLevel Drain valve parameters
	gModules[0].heads[0].fillLevelCylinderValve;
	fillLevelDrainValve[0].MpRecipeRegPar_0.PVName := ADR('gModules[0].heads[0]fillLevelDrainValve.parameters.machineData');
	fillLevelDrainValve[1].MpRecipeRegPar_0.PVName := ADR('gModules[0].heads[1].fillLevelDrainValve.parameters.machineData');
	fillLevelDrainValve[2].MpRecipeRegPar_0.PVName := ADR('gModules[1].heads[0].fillLevelDrainValve.parameters.machineData');
	fillLevelDrainValve[3].MpRecipeRegPar_0.PVName := ADR('gModules[1].heads[1].fillLevelDrainValve.parameters.machineData');

	FOR currentHead:=0 TO NUMBER_OF_HEADS_M1 DO
		fillLevelDrainValve[currentHead].MpRecipeRegPar_0.MpLink := ADR(gMachineRecipe);
		fillLevelDrainValve[currentHead].MpRecipeRegPar_0.Enable := TRUE;
		fillLevelDrainValve[currentHead].MpRecipeRegPar_0.Category := ADR(MACHINE_CATEGORY);
		fillLevelDrainValve[currentHead].MpRecipeRegPar_0();
	END_FOR

	fillLevelDrainValve[0].MpRecipeRegPar_1.PVName := ADR('gModules[0].heads[0].fillLevelDrainValve.parameters.processData');
	fillLevelDrainValve[1].MpRecipeRegPar_1.PVName := ADR('gModules[0].heads[1].fillLevelDrainValve.parameters.processData');
	fillLevelDrainValve[2].MpRecipeRegPar_1.PVName := ADR('gModules[1].heads[0].fillLevelDrainValve.parameters.processData');
	fillLevelDrainValve[3].MpRecipeRegPar_1.PVName := ADR('gModules[1].heads[1].fillLevelDrainValve.parameters.processData');

	FOR currentHead:=0 TO NUMBER_OF_HEADS_M1 DO
		fillLevelDrainValve[currentHead].MpRecipeRegPar_1.MpLink := ADR(gProcessRecipe);
		fillLevelDrainValve[currentHead].MpRecipeRegPar_1.Enable := TRUE;
		fillLevelDrainValve[currentHead].MpRecipeRegPar_1.Category := ADR(PROCESS_CATEGORY);
		fillLevelDrainValve[currentHead].MpRecipeRegPar_1();
	END_FOR

	FOR currentHead:=0 TO NUMBER_OF_HEADS_M1 DO

		pLocalValve ACCESS ADR(balanceTankValve[currentHead]);
		pLocalValve.valveName := gModules[getModuleIndex(currentHead)].heads[getHeadIndex(currentHead)].headName;
		strcat(ADR(pLocalValve.valveName), ADR(' Balance Tank Valve'));

		pLocalValve ACCESS ADR(fillValve[currentHead]);
		pLocalValve.valveName := gModules[getModuleIndex(currentHead)].heads[getHeadIndex(currentHead)].headName;
		strcat(ADR(pLocalValve.valveName), ADR(' Fill Valve'));

		pLocalValve ACCESS ADR(cylinderVentValve[currentHead]);
		pLocalValve.valveName := gModules[getModuleIndex(currentHead)].heads[getHeadIndex(currentHead)].headName;
		strcat(ADR(pLocalValve.valveName), ADR(' Cylinder Vent Valve'));

		pLocalValve ACCESS ADR(formingValve[currentHead]);
		pLocalValve.valveName := gModules[getModuleIndex(currentHead)].heads[getHeadIndex(currentHead)].headName;
		strcat(ADR(pLocalValve.valveName), ADR(' Forming Valve'));

        pLocalValve ACCESS ADR(nozzleValve[currentHead]);
        pLocalValve.valveName := gModules[getModuleIndex(currentHead)].heads[getHeadIndex(currentHead)].headName;
        strcat(ADR(pLocalValve.valveName), ADR(' Nozzle Valve'));

        pLocalValve ACCESS ADR(recirculationValve[currentHead]);
        pLocalValve.valveName := gModules[getModuleIndex(currentHead)].heads[getHeadIndex(currentHead)].headName;
        strcat(ADR(pLocalValve.valveName), ADR(' Recirculation Valve'));

        pLocalValve ACCESS ADR(sealPinValve[currentHead]);
        pLocalValve.valveName := gModules[getModuleIndex(currentHead)].heads[getHeadIndex(currentHead)].headName;
        strcat(ADR(pLocalValve.valveName), ADR(' Seal Pin Valve'));

        pLocalValve ACCESS ADR(counterStretchRodValve[currentHead]);
        pLocalValve.valveName := gModules[getModuleIndex(currentHead)].heads[getHeadIndex(currentHead)].headName;
        strcat(ADR(pLocalValve.valveName), ADR(' Counter Stretchrod Valve'));

		pLocalValve ACCESS ADR(fillLevelCylinderValve[currentHead]);
		pLocalValve.valveName := gModules[getModuleIndex(currentHead)].heads[getHeadIndex(currentHead)].headName;
		strcat(ADR(pLocalValve.valveName), ADR(' FillLevel Cylinder Valve'));

		pLocalValve ACCESS ADR(fillLevelSuctionValve[currentHead]);
		pLocalValve.valveName := gModules[getModuleIndex(currentHead)].heads[getHeadIndex(currentHead)].headName;
		strcat(ADR(pLocalValve.valveName), ADR(' FillLevel Suction Valve'));

		pLocalValve ACCESS ADR(fillLevelDrainValve[currentHead]);
		pLocalValve.valveName := gModules[getModuleIndex(currentHead)].heads[getHeadIndex(currentHead)].headName;
		strcat(ADR(pLocalValve.valveName), ADR(' FillLevel Drain Valve'));

    END_FOR

END_PROGRAM

PROGRAM _CYCLIC

	gMachineControl.commands.preformsEnteringMoldStart.CLK  := (gMachineControl.status.preformsEnteringMold = TRUE);
	gMachineControl.commands.preformsEnteringMoldStart();
	IF gMachineControl.commands.preformsEnteringMoldStart.Q = TRUE THEN
		FOR currentModule:=0 TO NUMBER_OF_MODULES_M1 DO
			FOR currentHead:=0 TO NUM_OF_HEADS_PER_MODULE_M1 DO
				IF ((gModules[currentModule].heads[currentHead].enable = TRUE) AND (gModules[currentModule].heads[currentHead].recirculationValve.status.errorActive <> TRUE)) THEN
					gModules[currentModule].heads[currentHead].recirculationValve.commands.open := FALSE;
					gModules[currentModule].heads[currentHead].recirculationValve.commands.close := TRUE;
				END_IF
			END_FOR
		END_FOR
	END_IF

    FOR currentModule:=0 TO NUMBER_OF_MODULES_M1 DO
        FOR currentHead:=0 TO NUM_OF_HEADS_PER_MODULE_M1 DO

            logArguments[0] := ADR(currentModule);
            logArguments[1] := ADR(currentHead);

            balanceTankAction;
            counterStretchRodAction;
            fillAction;
            cylinderVentAction;
            formingValveAction;
            nozzleAction;
            recirculationAction;
			sealPinAction;
			fillLevelCylinderValveAction;
			fillLevelSuctionValveAction;
			fillLevelDrainValveAction;

            IF (DiagCpuIsSimulated() = TRUE) THEN
                gModules[currentModule].heads[currentHead].fillValve.status.errorActive := FALSE;
                gModules[currentModule].heads[currentHead].formingValve.status.errorActive := FALSE;
                gModules[currentModule].heads[currentHead].recirculationValve.status.errorActive := FALSE;
                gModules[currentModule].heads[currentHead].sealPin.status.errorActive := FALSE;
                gModules[currentModule].heads[currentHead].nozzle.status.errorActive := FALSE;
                gModules[currentModule].heads[currentHead].cylinderVent.status.errorActive := FALSE;
				gModules[currentModule].heads[currentHead].counterStretchRod.status.errorActive := FALSE;
				gModules[currentModule].heads[currentHead].fillLevelCylinderValve.status.errorActive := FALSE;
				gModules[currentModule].heads[currentHead].fillLevelSuctionValve.status.errorActive := FALSE;
				gModules[currentModule].heads[currentHead].fillLevelDrainValve.status.errorActive := FALSE;

            END_IF

        END_FOR
    END_FOR

END_PROGRAM

PROGRAM _EXIT
	(* Insert code here *)

END_PROGRAM

(* ---- nozzleValve.st ---- *)
ACTION nozzleAction:

    pCurrentValve ACCESS ADR(gModules[currentModule].heads[currentHead].nozzle);
    pLocalValve ACCESS ADR(nozzleValve[indexOf(currentModule, currentHead, NUM_OF_HEADS_PER_MODULE)]);

	IF (pCurrentValve.parameters.machineData.enabled = TRUE) THEN
		IF (pCurrentValve.status.errorActive <> TRUE) THEN

			IF (((pCurrentValve.commands.open = TRUE) AND (pCurrentValve.commands.close = FALSE)) AND
				(pLocalValve.doOpen = FALSE)) THEN
				logDebug(pLocalValve.valveName, 'Module %h, Head %h, Open Command', ADR(logArguments));
				pLocalValve.doOpen := TRUE;
				pLocalValve.doClose := FALSE;
			END_IF

			IF (((pCurrentValve.commands.close = TRUE) AND (pCurrentValve.commands.open = FALSE)) AND
				(pLocalValve.doClose = FALSE)) THEN
				logDebug(pLocalValve.valveName, 'Module %h, Head %h, Close Command', ADR(logArguments));
				pLocalValve.doClose := TRUE;
				pLocalValve.doOpen := FALSE;
			END_IF

			IF (((pCurrentValve.commands.close = FALSE) AND (pCurrentValve.commands.open = FALSE)) AND
				((pLocalValve.doClose <> FALSE) OR (pLocalValve.doOpen <> FALSE))) THEN
				logDebug(pLocalValve.valveName, 'Module %h, Head %h, Center Command', ADR(logArguments));
				pLocalValve.doClose := FALSE;
				pLocalValve.doOpen := FALSE;
			END_IF

		END_IF

        checkValveAlarms;
        updateValveState;

		// 20ms debounce timer
		pLocalValve.openDebounceTimer.IN    := pLocalValve.diOpened;
		pLocalValve.openDebounceTimer.PT    := pCurrentValve.parameters.machineData.debounceTime;
		pLocalValve.openDebounceTimer();

		// 20ms debounce timer
		pLocalValve.closeDebounceTimer.IN := pLocalValve.diClosed;
		pLocalValve.closeDebounceTimer.PT := pCurrentValve.parameters.machineData.debounceTime;
		pLocalValve.closeDebounceTimer();

		pCurrentValve.status.opened             := pLocalValve.openDebounceTimer.Q;
		pCurrentValve.status.closed             := pLocalValve.closeDebounceTimer.Q;
		pCurrentValve.status.centered           := ((pCurrentValve.status.opened <> TRUE) AND (pCurrentValve.status.closed <> TRUE));
		pCurrentValve.status.position           := 0;
		pCurrentValve.status.fullFlowAchieved   := FALSE;

        handleValveErrors;

	END_IF

END_ACTION

(* ---- recirculationValve.st ---- *)
ACTION recirculationAction:
    pCurrentValve ACCESS ADR(gModules[currentModule].heads[currentHead].recirculationValve);
    pLocalValve ACCESS ADR(recirculationValve[indexOf(currentModule, currentHead, NUM_OF_HEADS_PER_MODULE)]);

	IF (pCurrentValve.parameters.machineData.enabled = TRUE) THEN
		IF (pCurrentValve.status.errorActive <> TRUE) THEN

			IF (((pCurrentValve.commands.open = TRUE) AND (pCurrentValve.commands.close = FALSE)) AND
				(pLocalValve.doOpen = FALSE)) THEN
				logDebug(pLocalValve.valveName, 'Module %h, Head %h, Open Command', ADR(logArguments));
				pLocalValve.doOpen  := TRUE;
				pLocalValve.doClose := FALSE;
			END_IF

			IF (((pCurrentValve.commands.close = TRUE) AND (pCurrentValve.commands.open = FALSE)) AND
				(pLocalValve.doClose = FALSE)) THEN
				logDebug(pLocalValve.valveName, 'Module %h, Head %h, Close Command', ADR(logArguments));
				pLocalValve.doOpen  := FALSE;
				pLocalValve.doClose := TRUE;
			END_IF

			IF (((pCurrentValve.commands.close = FALSE) AND (pCurrentValve.commands.open = FALSE)) AND
				((pLocalValve.doClose <> FALSE) OR (pLocalValve.doOpen <> FALSE))) THEN
				logDebug(pLocalValve.valveName, 'Module %h, Head %h, Center Command', ADR(logArguments));
				pLocalValve.doOpen := FALSE;
				pLocalValve.doClose := FALSE;
			END_IF

        END_IF

        checkValveAlarms;
        updateValveState;

		// 20ms debounce timer
		pLocalValve.openDebounceTimer.IN    := pLocalValve.diOpened;
		pLocalValve.openDebounceTimer.PT    := pCurrentValve.parameters.machineData.debounceTime;
		pLocalValve.openDebounceTimer();

		// 20ms debounce timer
		pLocalValve.closeDebounceTimer.IN := pLocalValve.diClosed;
		pLocalValve.closeDebounceTimer.PT := pCurrentValve.parameters.machineData.debounceTime;
		pLocalValve.closeDebounceTimer();

		pCurrentValve.status.opened             := pLocalValve.openDebounceTimer.Q;
		pCurrentValve.status.closed             := pLocalValve.closeDebounceTimer.Q;
		pCurrentValve.status.centered           := ((pCurrentValve.status.opened <> TRUE) AND (pCurrentValve.status.closed <> TRUE));
		pCurrentValve.status.position           := 0;
		pCurrentValve.status.fullFlowAchieved   := FALSE;

        handleValveErrors;

	END_IF

END_ACTION

(* ---- sealPinValve.st ---- *)
ACTION sealPinAction:

	pCurrentValve ACCESS ADR(gModules[currentModule].heads[currentHead].sealPin);
	pLocalValve ACCESS ADR(sealPinValve[indexOf(currentModule, currentHead, NUM_OF_HEADS_PER_MODULE)]);

	IF (pCurrentValve.parameters.machineData.enabled = TRUE) THEN
		IF (pCurrentValve.status.errorActive <> TRUE) THEN

			IF (((pCurrentValve.commands.open = TRUE) AND (pCurrentValve.commands.close = FALSE)) AND
				(pLocalValve.doOpen = FALSE)) THEN
				logDebug(pLocalValve.valveName, 'Module %h, Head %h, Open Command', ADR(logArguments));
				pLocalValve.doOpen := TRUE;
				pLocalValve.doClose := FALSE;
			END_IF

			IF (((pCurrentValve.commands.close = TRUE) AND (pCurrentValve.commands.open = FALSE)) AND
				(pLocalValve.doClose = FALSE)) THEN
				logDebug(pLocalValve.valveName, 'Module %h, Head %h, Close Command', ADR(logArguments));
				pLocalValve.doClose := TRUE;
				pLocalValve.doOpen := FALSE;
			END_IF

			IF (((pCurrentValve.commands.close = FALSE) AND (pCurrentValve.commands.open = FALSE)) AND
				((pLocalValve.doClose <> FALSE) OR (pLocalValve.doOpen <> FALSE))) THEN
				logDebug(pLocalValve.valveName, 'Module %h, Head %h, Center Command', ADR(logArguments));
				pLocalValve.doClose := FALSE;
				pLocalValve.doOpen := FALSE;
			END_IF

		END_IF

		IF (pCurrentValve.status.position >= pCurrentValve.parameters.machineData.fullFlowPosition) THEN
			pCurrentValve.status.fullFlowAchieved := TRUE;
		ELSE
			pCurrentValve.status.fullFlowAchieved := FALSE;
		END_IF

		IF (pCurrentValve.status.position >= pCurrentValve.parameters.machineData.fullOpenPosition) THEN
			pCurrentValve.status.fullOpenedPosition := TRUE;
		ELSE
			pCurrentValve.status.fullOpenedPosition := FALSE;
		END_IF
		pLocalValve.diOpened := pCurrentValve.status.fullOpenedPosition;

		IF (pCurrentValve.status.position <= pCurrentValve.parameters.machineData.fullClosedPosition) THEN
			pLocalValve.diClosed := TRUE;
		ELSE
			pLocalValve.diClosed := FALSE;
		END_IF

        checkValveAlarms;
        updateValveState;

		// 20ms debounce timer
		pLocalValve.openDebounceTimer.IN    := pLocalValve.diOpened;
		pLocalValve.openDebounceTimer.PT    := pCurrentValve.parameters.machineData.debounceTime;
		pLocalValve.openDebounceTimer();

		// 20ms debounce timer
		pLocalValve.closeDebounceTimer.IN := pLocalValve.diClosed;
		pLocalValve.closeDebounceTimer.PT := pCurrentValve.parameters.machineData.debounceTime;
		pLocalValve.closeDebounceTimer();

		pCurrentValve.status.opened         := pLocalValve.openDebounceTimer.Q;
		pCurrentValve.status.closed         := pLocalValve.closeDebounceTimer.Q;
		pCurrentValve.status.centered       := ((pCurrentValve.status.opened <> TRUE) AND (pCurrentValve.status.closed <> TRUE));
		pCurrentValve.status.position       := (pLocalValve.position - pCurrentValve.parameters.machineData.scalingOffset) * pCurrentValve.parameters.machineData.scalingFactor;

        handleValveErrors;

	END_IF

END_ACTION

(* ---- valveAlarms.st ---- *)
// common code for handling valve alarms
// pLocalValve, pCurrentValve must be set to an valid point before the action is called
ACTION checkValveAlarms:

    IF ((ADR(pLocalValve) <> 0) AND (ADR(pCurrentValve) <> 0)) THEN

        // ensure that the valve opens
        pLocalValve.openErrorTimer.IN    := ((pCurrentValve.commands.open = TRUE) AND (pLocalValve.diOpened = FALSE));
        pLocalValve.openErrorTimer.PT    := pCurrentValve.parameters.machineData.timeout;
        pLocalValve.openErrorTimer();

        IF pLocalValve.openErrorTimer.IN = TRUE THEN
            pCurrentValve.status.openTime :=	TIME_TO_REAL(pLocalValve.openErrorTimer.ET) / 1000.0;
        END_IF

        // ensure that the valve closes
        pLocalValve.closeErrorTimer.IN := ((pCurrentValve.commands.close = TRUE) AND (pLocalValve.diClosed = FALSE));
        pLocalValve.closeErrorTimer.PT := pCurrentValve.parameters.machineData.timeout;
        pLocalValve.closeErrorTimer();

        IF pLocalValve.closeErrorTimer.IN = TRUE THEN
            pCurrentValve.status.closeTime :=	TIME_TO_REAL(pLocalValve.closeErrorTimer.ET) / 1000.0;
        END_IF

        pLocalValve.openError_r_trig.CLK := pLocalValve.openErrorTimer.Q;
        pLocalValve.openError_r_trig();
        IF (pLocalValve.openError_r_trig.Q = TRUE) THEN
            valveErrorName := pLocalValve.valveName;
            logError(pLocalValve.valveName, 'Module %h, Head %h, valve did not open', ADR(logArguments));
            IF (pLocalValve.openAlarmID = 0) THEN
                pLocalValve.openAlarmID                := MpAlarmXSet(gAlarmXCore, 'VALVE_NOT_OPENED');
            ELSE
                logError(pLocalValve.valveName, 'Module %h, Head %h, valve did not open occurred when alarm already active', ADR(logArguments));
            END_IF

        END_IF

        pLocalValve.closeError_r_trig.CLK := pLocalValve.closeErrorTimer.Q;
        pLocalValve.closeError_r_trig();
        IF (pLocalValve.closeError_r_trig.Q = TRUE) THEN
            valveErrorName := pLocalValve.valveName;
            logError(pLocalValve.valveName, 'Module %h, Head %h, valve did not close', ADR(logArguments));
            IF (pLocalValve.closeAlarmID = 0) THEN
                pLocalValve.closeAlarmID                 := MpAlarmXSet(gAlarmXCore, 'VALVE_NOT_CLOSED');
            ELSE
                logError(pLocalValve.valveName, 'Module %h, Head %h, valve did not close occurred when alarm already active', ADR(logArguments));
            END_IF
        END_IF

        pLocalValve.open_and_close_error_r_trig.CLK := ((pCurrentValve.commands.open = TRUE) AND (pCurrentValve.commands.close = TRUE));
        pLocalValve.open_and_close_error_r_trig();
        IF (pLocalValve.open_and_close_error_r_trig.Q = TRUE) THEN
            valveErrorName      := pLocalValve.valveName;
            logError(pLocalValve.valveName, 'Module %h, Head %h, valve commanded open and close', ADR(logArguments));
            IF (pLocalValve.openAndCloseAlarmID = 0) THEN
                pLocalValve.openAndCloseAlarmID                 := MpAlarmXSet(gAlarmXCore, 'VALVE_COMMANDED_OPEN_AND_CLOSE');
            ELSE
                logError(pLocalValve.valveName, 'Module %h, Head %h, valve commanded open and close occurred when alarm already active', ADR(logArguments));
            END_IF
        END_IF

        pLocalValve.powerOnTimer.IN := gMachineControl.commands.powerOn;
        pLocalValve.powerOnTimer.PT := T#5s;
        pLocalValve.powerOnTimer();

        pLocalValve.io_error_r_trig.CLK := ((pLocalValve.inputModuleOk = FALSE) OR (pLocalValve.outputModuleOk = FALSE)) AND (pLocalValve.powerOnTimer.Q = TRUE);
        pLocalValve.io_error_r_trig();
        IF (pLocalValve.io_error_r_trig.Q = TRUE) THEN
            valveErrorName      := pLocalValve.valveName;
            logError(pLocalValve.valveName, 'Module %h, Head %h, valve io missing', ADR(logArguments));
            IF (pLocalValve.moduleOKAlarmID = 0) THEN
                pLocalValve.moduleOKAlarmID         := MpAlarmXSet(gAlarmXCore, 'VALVE_IO_MISSING');
            ELSE
                logError(pLocalValve.valveName, 'Module %h, Head %h, valve io missing occurred when alarm already active', ADR(logArguments));
            END_IF
        END_IF

        pLocalValve.io_error_f_trig.CLK := ((pLocalValve.inputModuleOk = FALSE) OR (pLocalValve.outputModuleOk = FALSE));
        pLocalValve.io_error_f_trig();
        IF (pLocalValve.io_error_f_trig.Q = TRUE) THEN
            MpAlarmXResetID(gAlarmXCore, pLocalValve.moduleOKAlarmID);
            pLocalValve.moduleOKAlarmID         := 0;
        END_IF
    END_IF

END_ACTION

ACTION handleValveErrors:

    IF ((ADR(pLocalValve) <> 0) AND (ADR(pCurrentValve) <> 0)) THEN

        pCurrentValve.status.errorActive        := ((pLocalValve.openAlarmID <> 0) OR (pLocalValve.closeAlarmID <> 0) OR (pLocalValve.openAndCloseAlarmID <> 0) OR (pLocalValve.moduleOKAlarmID <> 0));

        IF (pCurrentValve.status.errorActive = TRUE) THEN
            pCurrentValve.commands.close            := FALSE;
            pCurrentValve.commands.open             := FALSE;
        END_IF
        IF (pCurrentValve.commands.errorAcknowledge = TRUE) THEN
            pCurrentValve.commands.errorAcknowledge := FALSE;
            pCurrentValve.status.errorActive        := FALSE;

            IF (pLocalValve.openAlarmID <> 0) THEN
                logError(pLocalValve.valveName, 'Module %h, Head %h, Acknowledging Error', ADR(logArguments));
                IF (MpAlarmXResetID(gAlarmXCore, pLocalValve.openAlarmID) <> 0) THEN
                    logError(pLocalValve.valveName, 'Module %h, Head %h, Could not acknowledge alarm with ID, resetting all OPENED alarms', ADR(logArguments));
                    MpAlarmXReset(gAlarmXCore, 'VALVE_NOT_OPENED');
                END_IF
                pLocalValve.openAlarmID := 0;
            END_IF

            IF (pLocalValve.closeAlarmID <> 0) THEN
                logError(pLocalValve.valveName, 'Module %h, Head %h, Acknowledging Error', ADR(logArguments));
                IF (MpAlarmXResetID(gAlarmXCore, pLocalValve.closeAlarmID) <> 0) THEN
                    logError(pLocalValve.valveName, 'Module %h, Head %h, Could not acknowledge alarm with ID, resetting all CLOSED alarms', ADR(logArguments));
                    MpAlarmXReset(gAlarmXCore, 'VALVE_NOT_CLOSED');
                END_IF
                pLocalValve.closeAlarmID := 0;
            END_IF

            IF (pLocalValve.openAndCloseAlarmID <> 0) THEN
                logError(pLocalValve.valveName, 'Module %h, Head %h, Acknowledging Error', ADR(logArguments));
                IF (MpAlarmXResetID(gAlarmXCore, pLocalValve.openAndCloseAlarmID) <> 0) THEN
                    logError(pLocalValve.valveName, 'Module %h, Head %h, Could not acknowledge alarm with ID, resetting all OPEN_AND_CLOSE alarms', ADR(logArguments));
                    MpAlarmXReset(gAlarmXCore, 'VALVE_COMMANDED_OPEN_AND_CLOSE');
                END_IF
                pLocalValve.openAndCloseAlarmID := 0;
            END_IF
        END_IF
    END_IF

END_ACTION

ACTION updateValveState:

    IF ((ADR(pLocalValve) <> 0) AND (ADR(pCurrentValve) <> 0)) THEN

		//Set ValveState integer value for grphics
		pCurrentValve.status.valveState := 0;
		IF pLocalValve.doOpen = FALSE AND pLocalValve.diOpened = FALSE THEN
			pCurrentValve.status.valveState := 1;
		ELSIF pLocalValve.doOpen = TRUE AND pLocalValve.diOpened = FALSE THEN
			pCurrentValve.status.valveState := 2;
		ELSIF pLocalValve.doOpen = TRUE AND pLocalValve.diOpened = TRUE THEN
			pCurrentValve.status.valveState := 3;
		ELSIF pLocalValve.doOpen = FALSE AND pLocalValve.diOpened = TRUE THEN
			pCurrentValve.status.valveState := 4;
		ELSIF pLocalValve.doClose = FALSE AND pLocalValve.diClosed = FALSE THEN
			pCurrentValve.status.valveState := 5;
		ELSIF pLocalValve.doClose = TRUE AND pLocalValve.diClosed = FALSE THEN
			pCurrentValve.status.valveState := 6;
		ELSIF pLocalValve.doClose = TRUE AND pLocalValve.diClosed = TRUE THEN
			pCurrentValve.status.valveState := 7;
		ELSIF pLocalValve.doClose = FALSE AND pLocalValve.diClosed = TRUE THEN
			pCurrentValve.status.valveState := 8;
		END_IF

    END_IF

END_ACTION
